PROGRAM Instanziierung
VAR
	Skill		:BasisSkill;
	TestSkill	:TestSkill_1;
END_VAR

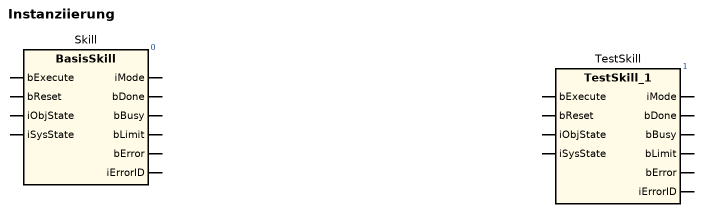
Skill(); // BasisSkill
TestSkill(); // TestSkill_1

END_PROGRAM

(* stored: Version 1.1.0.1
   POU Instanziierung: Id {9a254260-5048-4e24-b6bc-dec306593a6c}, SpecialFunc None *)
